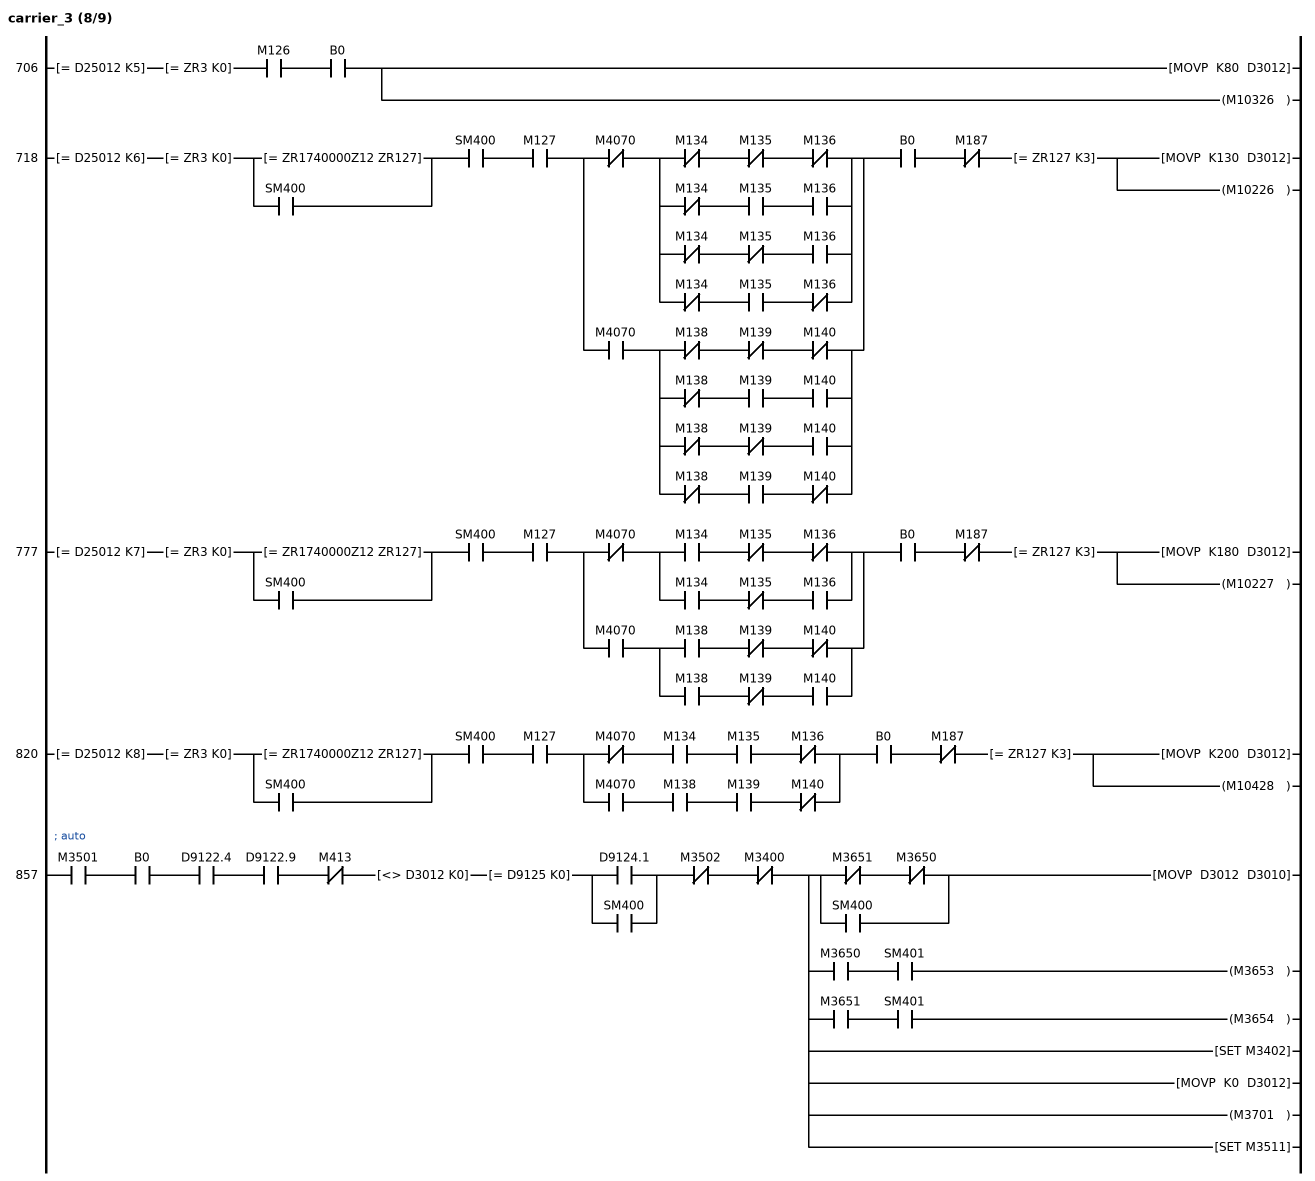
[picture p72: ladder of carrier_3, rungs at steps 706 to 857]
706   LD=     D25012 K5
      AND=    ZR3 K0
      AND     M126
      AND     B0
      MOVP    K80 D3012
      OUT     M10326
718   LD=     D25012 K6
      AND=    ZR3 K0
      LD=     ZR1740000Z12 ZR127
      OR      SM400
      ANB
      AND     SM400
      AND     M127
      LDI     M4070
      LDI     M134
      ANI     M135
      ANI     M136
      LDI     M134
      AND     M135
      AND     M136
      ORB
      LDI     M134
      ANI     M135
      AND     M136
      ORB
      LDI     M134
      AND     M135
      ANI     M136
      ORB
      ANB
      LD      M4070
      LDI     M138
      ANI     M139
      ANI     M140
      LDI     M138
      AND     M139
      AND     M140
      ORB
      LDI     M138
      ANI     M139
      AND     M140
      ORB
      LDI     M138
      AND     M139
      ANI     M140
      ORB
      ANB
      ORB
      ANB
      AND     B0
      ANI     M187
      AND=    ZR127 K3
      MOVP    K130 D3012
      OUT     M10226
777   LD=     D25012 K7
      AND=    ZR3 K0
      LD=     ZR1740000Z12 ZR127
      OR      SM400
      ANB
      AND     SM400
      AND     M127
      LDI     M4070
      LD      M134
      ANI     M135
      ANI     M136
      LD      M134
      ANI     M135
      AND     M136
      ORB
      ANB
      LD      M4070
      LD      M138
      ANI     M139
      ANI     M140
      LD      M138
      ANI     M139
      AND     M140
      ORB
      ANB
      ORB
      ANB
      AND     B0
      ANI     M187
      AND=    ZR127 K3
      MOVP    K180 D3012
      OUT     M10227
820   LD=     D25012 K8
      AND=    ZR3 K0
      LD=     ZR1740000Z12 ZR127
      OR      SM400
      ANB
      AND     SM400
      AND     M127
      LDI     M4070
      AND     M134
      AND     M135
      ANI     M136
      LD      M4070
      AND     M138
      AND     M139
      ANI     M140
      ORB
      ANB
      AND     B0
      ANI     M187
      AND=    ZR127 K3
      MOVP    K200 D3012
      OUT     M10428
; auto
857   LD      M3501
      AND     B0
      AND     D9122.4
      AND     D9122.9
      ANI     M413
      AND<>   D3012 K0
      AND=    D9125 K0
      LD      D9124.1
      OR      SM400
      ANB
      ANI     M3502
      ANI     M3400
      MPS
      LDI     M3651
      ANI     M3650
      OR      SM400
      ANB
      MOVP    D3012 D3010
      MRD
      AND     M3650
      AND     SM401
      OUT     M3653
      MRD
      AND     M3651
      AND     SM401
      OUT     M3654
      MPP
      SET     M3402
      MOVP    K0 D3012
      OUT     M3701
      SET     M3511
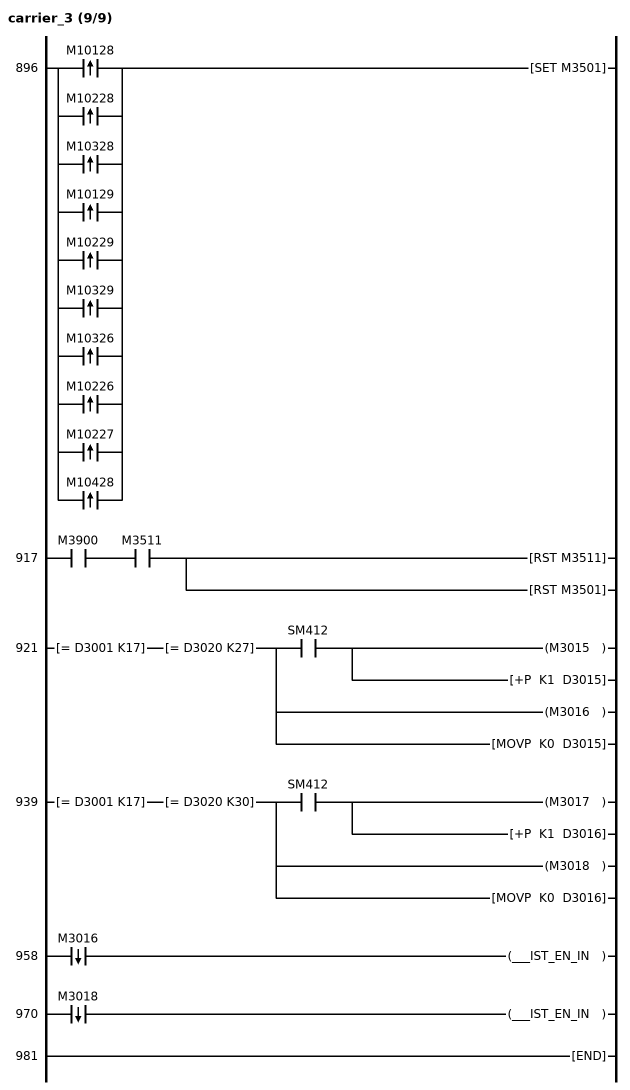
896   LDP     M10128
      ORP     M10228
      ORP     M10328
      ORP     M10129
      ORP     M10229
      ORP     M10329
      ORP     M10326
      ORP     M10226
      ORP     M10227
      ORP     M10428
      SET     M3501
917   LD      M3900
      AND     M3511
      RST     M3511
      RST     M3501
921   LD=     D3001 K17
      AND=    D3020 K27
      MPS
      AND     SM412
      OUT     M3015
      +P      K1 D3015
      MPP
      OUT     M3016
      MOVP    K0 D3015
939   LD=     D3001 K17
      AND=    D3020 K30
      MPS
      AND     SM412
      OUT     M3017
      +P      K1 D3016
      MPP
      OUT     M3018
      MOVP    K0 D3016
; FB BLK START I+ST_76367eaf8b844e8d(__IST_76367eaf8b844e8d)
958   LDF     M3016
      OUT     ___IST_EN_IN
; FB START
; FB_NAME I+ST_76367eaf8b844e8d
; INSTANCE_NAME __IST_76367eaf8b844e8d
; FB IN_B:__IST_EN_IN
; FB OUT___IST_EN_OUT:B
; FB END
; FB BLK END
; FB BLK START I+ST_4f96081e274e4d1c(__IST_4f96081e274e4d1c)
970   LDF     M3018
      OUT     ___IST_EN_IN
; FB START
; FB_NAME I+ST_4f96081e274e4d1c
; INSTANCE_NAME __IST_4f96081e274e4d1c
; FB IN_B:__IST_EN_IN
; FB OUT___IST_EN_OUT:B
; FB END
; FB BLK END
981   END
END_PROGRAM

PROGRAM carrier_4
VAR
  c_comm_4 : c_comm_4;
END_VAR
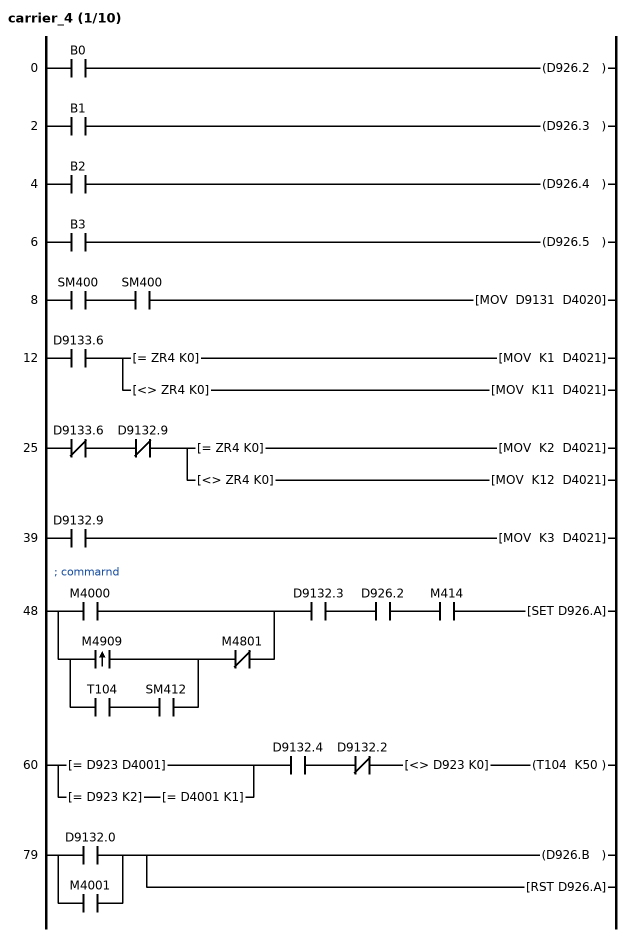
0     LD      B0
      OUT     D926.2
2     LD      B1
      OUT     D926.3
4     LD      B2
      OUT     D926.4
6     LD      B3
      OUT     D926.5
8     LD      SM400
      AND     SM400
      MOV     D9131 D4020
12    LD      D9133.6
      MPS
      AND=    ZR4 K0
      MOV     K1 D4021
      MPP
      AND<>   ZR4 K0
      MOV     K11 D4021
25    LDI     D9133.6
      ANI     D9132.9
      MPS
      AND=    ZR4 K0
      MOV     K2 D4021
      MPP
      AND<>   ZR4 K0
      MOV     K12 D4021
39    LD      D9132.9
      MOV     K3 D4021
; commarnd
48    LD      M4000
      LDP     M4909
      LD      T104
      AND     SM412
      ORB
      ANI     M4801
      ORB
      AND     D9132.3
      AND     D926.2
      AND     M414
      SET     D926.A
60    LD=     D923 D4001
      LD=     D923 K2
      AND=    D4001 K1
      ORB
      AND     D9132.4
      ANI     D9132.2
      AND<>   D923 K0
      OUT     T104 K50
79    LD      D9132.0
      OR      M4001
      OUT     D926.B
      RST     D926.A
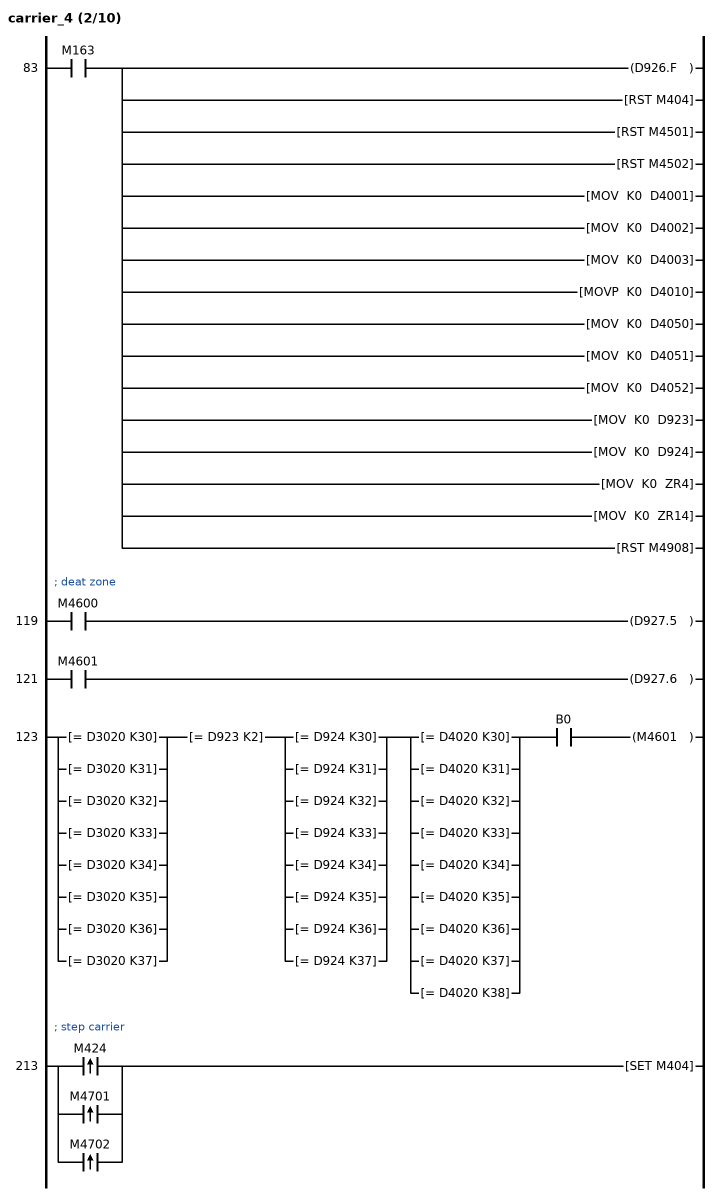
83    LD      M163
      OUT     D926.F
      RST     M404
      RST     M4501
      RST     M4502
      MOV     K0 D4001
      MOV     K0 D4002
      MOV     K0 D4003
      MOVP    K0 D4010
      MOV     K0 D4050
      MOV     K0 D4051
      MOV     K0 D4052
      MOV     K0 D923
      MOV     K0 D924
      MOV     K0 ZR4
      MOV     K0 ZR14
      RST     M4908
; deat zone
119   LD      M4600
      OUT     D927.5
121   LD      M4601
      OUT     D927.6
123   LD=     D3020 K30
      OR=     D3020 K31
      OR=     D3020 K32
      OR=     D3020 K33
      OR=     D3020 K34
      OR=     D3020 K35
      OR=     D3020 K36
      OR=     D3020 K37
      AND=    D923 K2
      LD=     D924 K30
      OR=     D924 K31
      OR=     D924 K32
      OR=     D924 K33
      OR=     D924 K34
      OR=     D924 K35
      OR=     D924 K36
      OR=     D924 K37
      ANB
      LD=     D4020 K30
      OR=     D4020 K31
      OR=     D4020 K32
      OR=     D4020 K33
      OR=     D4020 K34
      OR=     D4020 K35
      OR=     D4020 K36
      OR=     D4020 K37
      OR=     D4020 K38
      ANB
      AND     B0
      OUT     M4601
; step carrier
213   LDP     M424
      ORP     M4701
      ORP     M4702
      SET     M404
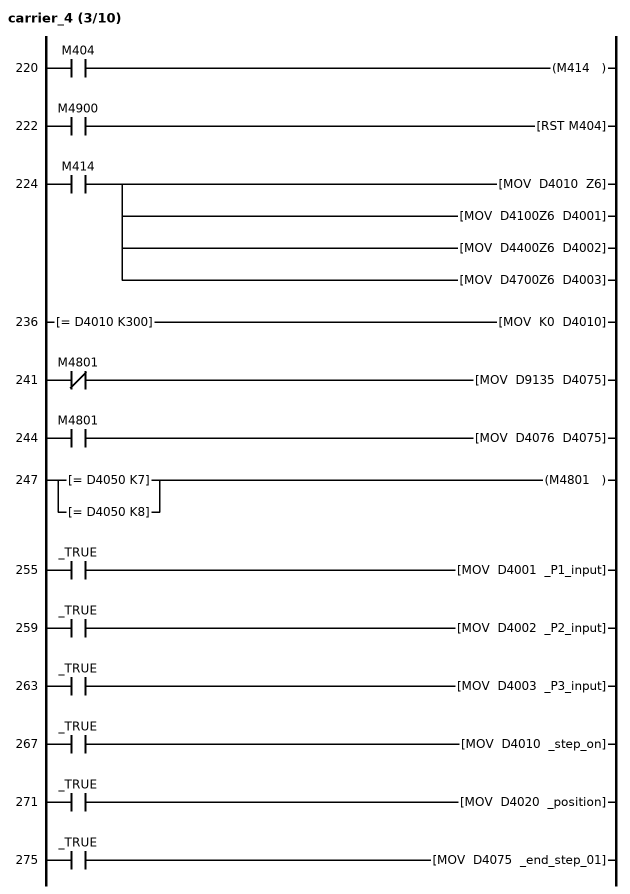
220   LD      M404
      OUT     M414
222   LD      M4900
      RST     M404
224   LD      M414
      MOV     D4010 Z6
      MOV     D4100Z6 D4001
      MOV     D4400Z6 D4002
      MOV     D4700Z6 D4003
236   LD=     D4010 K300
      MOV     K0 D4010
241   LDI     M4801
      MOV     D9135 D4075
244   LD      M4801
      MOV     D4076 D4075
247   LD=     D4050 K7
      OR=     D4050 K8
      OUT     M4801
; FB BLK START c_comm_4(c_comm_4)
255   LD      _TRUE
      MOV     D4001 _P1_input
259   LD      _TRUE
      MOV     D4002 _P2_input
263   LD      _TRUE
      MOV     D4003 _P3_input
267   LD      _TRUE
      MOV     D4010 _step_on
271   LD      _TRUE
      MOV     D4020 _position
275   LD      _TRUE
      MOV     D4075 _end_step_01
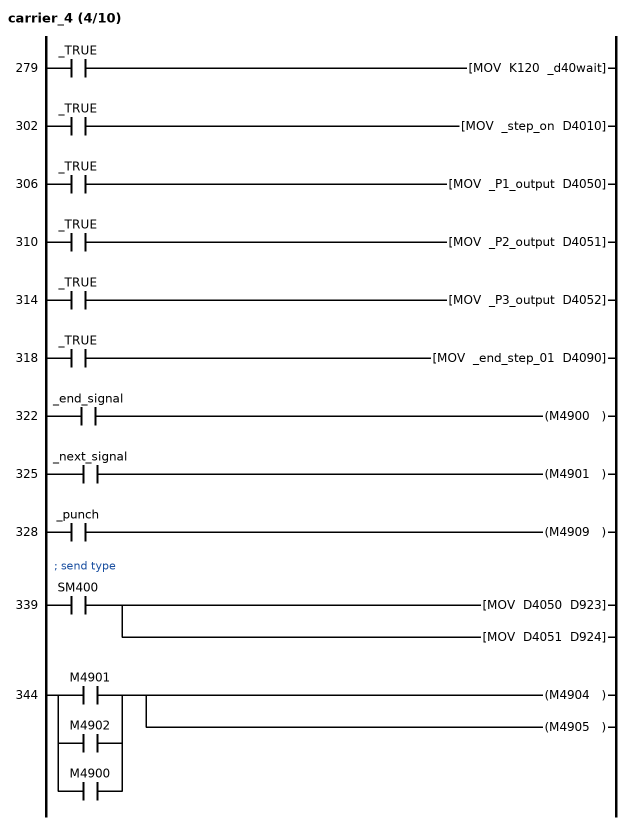
279   LD      _TRUE
      MOV     K120 _d40wait
; FB START
; FB_NAME c_comm_4
; INSTANCE_NAME c_comm_4
; FB IN_W:P1_input
; FB OUT_step_on:W
; FB IN_W:P2_input
; FB OUT_P1_output:W
; FB IN_W:P3_input
; FB OUT_P2_output:W
; FB IN_W:step_on
; FB OUT_P3_output:W
; FB IN_W:position
; FB OUT_end_step_01:W
; FB IN_W:end_step_01
; FB OUT_end_signal:B
; FB IN_W:d40wait
; FB OUT_next_signal:B
; FB OUT_punch:B
; FB END
302   LD      _TRUE
      MOV     _step_on D4010
306   LD      _TRUE
      MOV     _P1_output D4050
310   LD      _TRUE
      MOV     _P2_output D4051
314   LD      _TRUE
      MOV     _P3_output D4052
318   LD      _TRUE
      MOV     _end_step_01 D4090
322   LD      _end_signal
      OUT     M4900
325   LD      _next_signal
      OUT     M4901
328   LD      _punch
      OUT     M4909
; FB BLK END
; send type
339   LD      SM400
      MOV     D4050 D923
      MOV     D4051 D924
344   LD      M4901
      OR      M4902
      OR      M4900
      OUT     M4904
      OUT     M4905
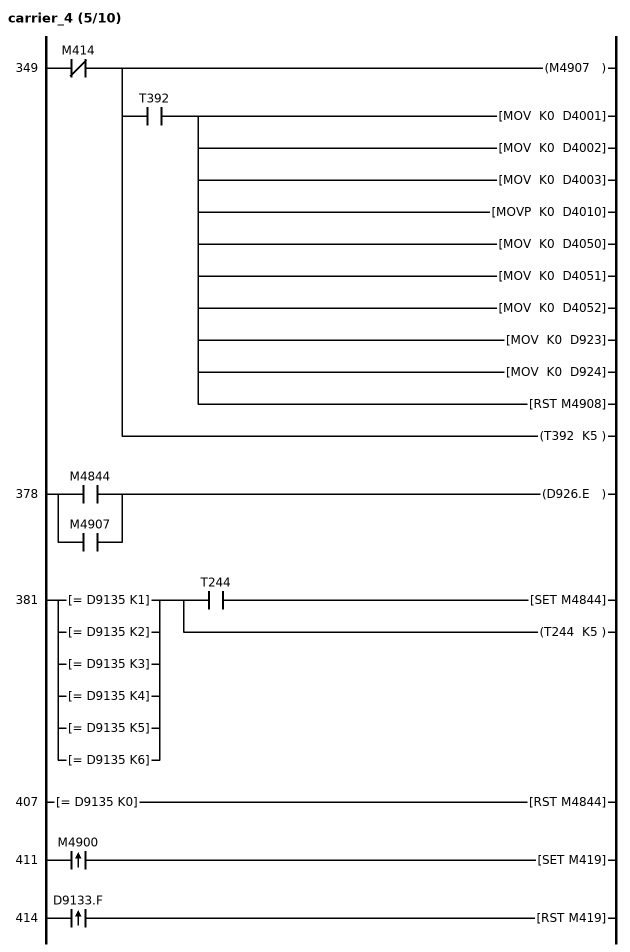
349   LDI     M414
      OUT     M4907
      MPS
      AND     T392
      MOV     K0 D4001
      MOV     K0 D4002
      MOV     K0 D4003
      MOVP    K0 D4010
      MOV     K0 D4050
      MOV     K0 D4051
      MOV     K0 D4052
      MOV     K0 D923
      MOV     K0 D924
      RST     M4908
      MPP
      OUT     T392 K5
378   LD      M4844
      OR      M4907
      OUT     D926.E
381   LD=     D9135 K1
      OR=     D9135 K2
      OR=     D9135 K3
      OR=     D9135 K4
      OR=     D9135 K5
      OR=     D9135 K6
      MPS
      AND     T244
      SET     M4844
      MPP
      OUT     T244 K5
407   LD=     D9135 K0
      RST     M4844
411   LDP     M4900
      SET     M419
414   LDP     D9133.F
      RST     M419
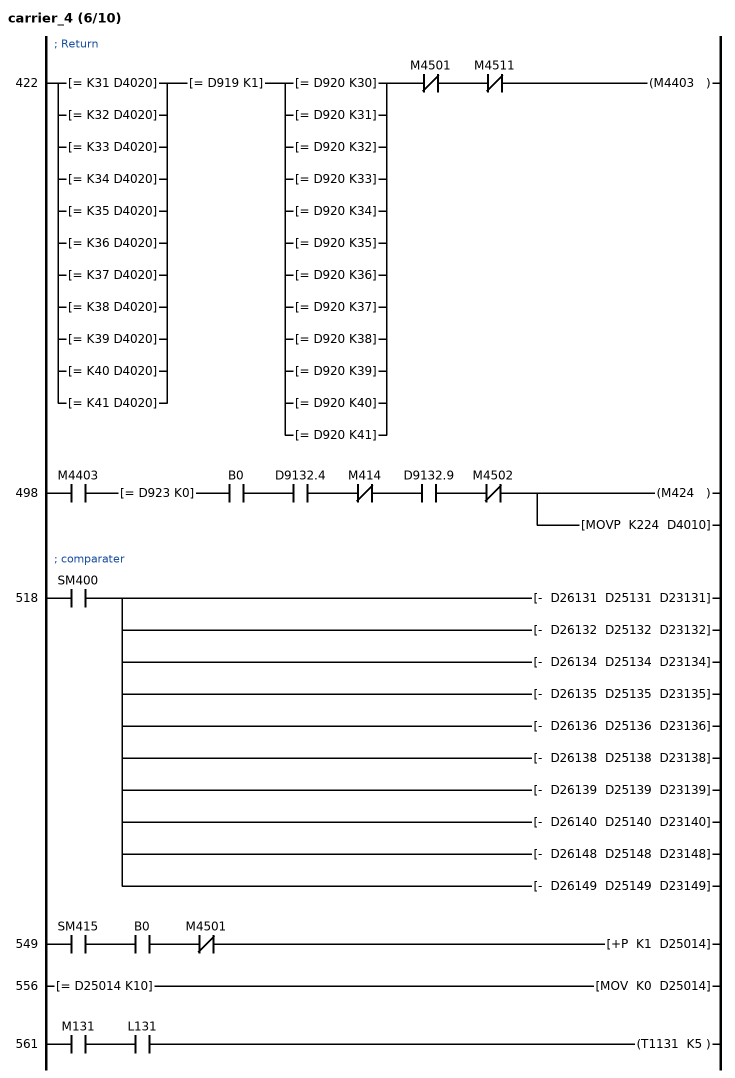
; Return
422   LD=     K31 D4020
      OR=     K32 D4020
      OR=     K33 D4020
      OR=     K34 D4020
      OR=     K35 D4020
      OR=     K36 D4020
      OR=     K37 D4020
      OR=     K38 D4020
      OR=     K39 D4020
      OR=     K40 D4020
      OR=     K41 D4020
      AND=    D919 K1
      LD=     D920 K30
      OR=     D920 K31
      OR=     D920 K32
      OR=     D920 K33
      OR=     D920 K34
      OR=     D920 K35
      OR=     D920 K36
      OR=     D920 K37
      OR=     D920 K38
      OR=     D920 K39
      OR=     D920 K40
      OR=     D920 K41
      ANB
      ANI     M4501
      ANI     M4511
      OUT     M4403
498   LD      M4403
      AND=    D923 K0
      AND     B0
      AND     D9132.4
      ANI     M414
      AND     D9132.9
      ANI     M4502
      OUT     M424
      MOVP    K224 D4010
; comparater
518   LD      SM400
      -       D26131 D25131 D23131
      -       D26132 D25132 D23132
      -       D26134 D25134 D23134
      -       D26135 D25135 D23135
      -       D26136 D25136 D23136
      -       D26138 D25138 D23138
      -       D26139 D25139 D23139
      -       D26140 D25140 D23140
      -       D26148 D25148 D23148
      -       D26149 D25149 D23149
549   LD      SM415
      AND     B0
      ANI     M4501
      +P      K1 D25014
556   LD=     D25014 K10
      MOV     K0 D25014
561   LD      M131
      AND     L131
      OUT     T1131 K5
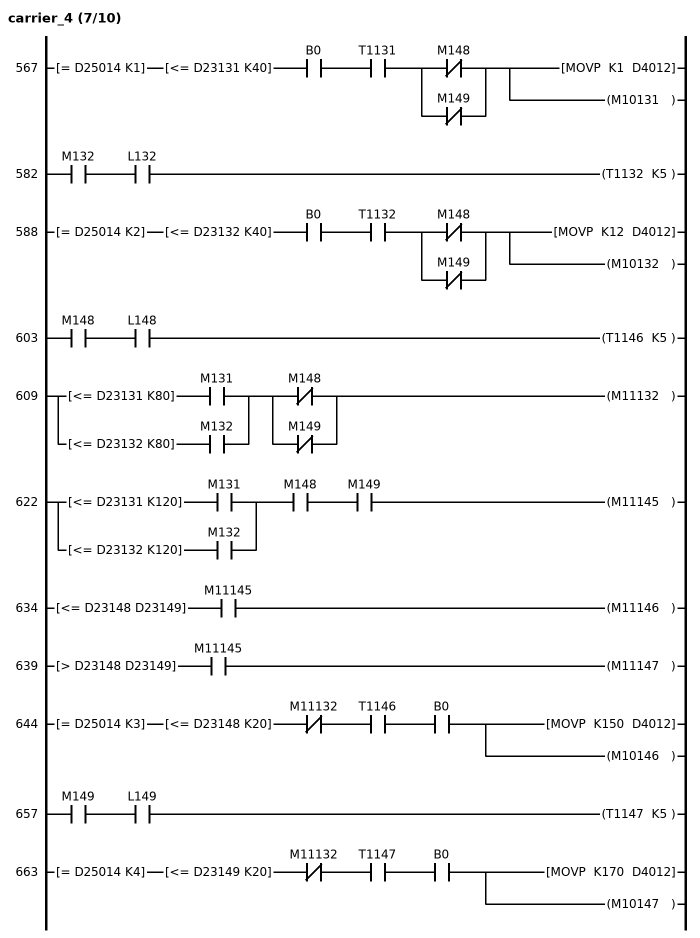
567   LD=     D25014 K1
      AND<=   D23131 K40
      AND     B0
      AND     T1131
      LDI     M148
      ORI     M149
      ANB
      MOVP    K1 D4012
      OUT     M10131
582   LD      M132
      AND     L132
      OUT     T1132 K5
588   LD=     D25014 K2
      AND<=   D23132 K40
      AND     B0
      AND     T1132
      LDI     M148
      ORI     M149
      ANB
      MOVP    K12 D4012
      OUT     M10132
603   LD      M148
      AND     L148
      OUT     T1146 K5
609   LD<=    D23131 K80
      AND     M131
      LD<=    D23132 K80
      AND     M132
      ORB
      LDI     M148
      ORI     M149
      ANB
      OUT     M11132
622   LD<=    D23131 K120
      AND     M131
      LD<=    D23132 K120
      AND     M132
      ORB
      AND     M148
      AND     M149
      OUT     M11145
634   LD<=    D23148 D23149
      AND     M11145
      OUT     M11146
639   LD>     D23148 D23149
      AND     M11145
      OUT     M11147
644   LD=     D25014 K3
      AND<=   D23148 K20
      ANI     M11132
      AND     T1146
      AND     B0
      MOVP    K150 D4012
      OUT     M10146
657   LD      M149
      AND     L149
      OUT     T1147 K5
663   LD=     D25014 K4
      AND<=   D23149 K20
      ANI     M11132
      AND     T1147
      AND     B0
      MOVP    K170 D4012
      OUT     M10147
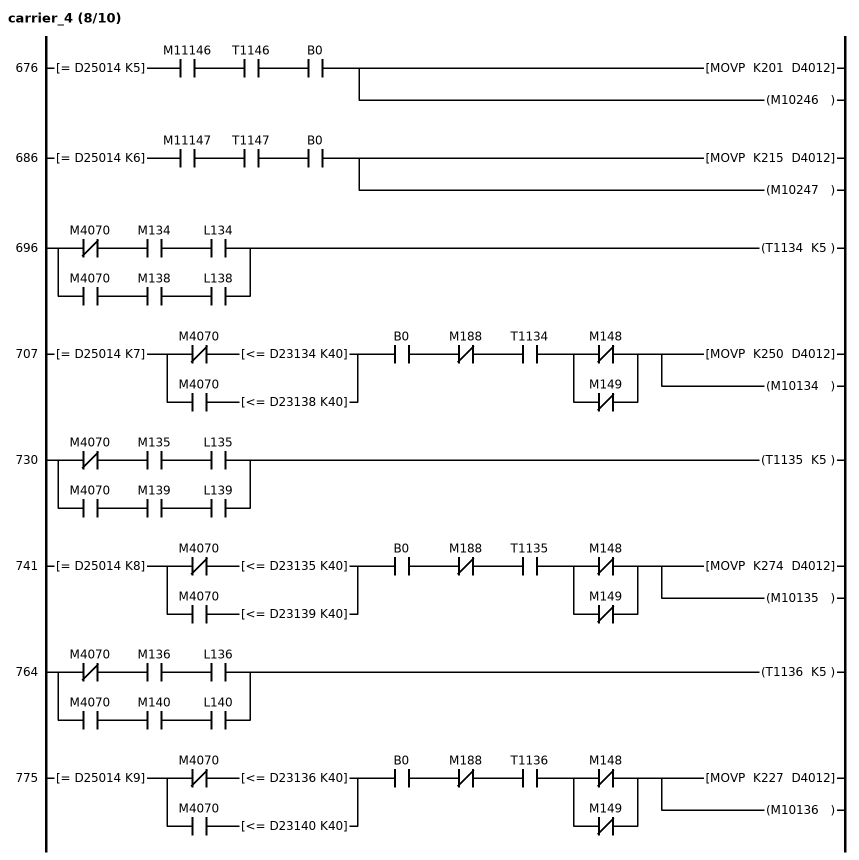
676   LD=     D25014 K5
      AND     M11146
      AND     T1146
      AND     B0
      MOVP    K201 D4012
      OUT     M10246
686   LD=     D25014 K6
      AND     M11147
      AND     T1147
      AND     B0
      MOVP    K215 D4012
      OUT     M10247
696   LDI     M4070
      AND     M134
      AND     L134
      LD      M4070
      AND     M138
      AND     L138
      ORB
      OUT     T1134 K5
707   LD=     D25014 K7
      LDI     M4070
      AND<=   D23134 K40
      LD      M4070
      AND<=   D23138 K40
      ORB
      ANB
      AND     B0
      ANI     M188
      AND     T1134
      LDI     M148
      ORI     M149
      ANB
      MOVP    K250 D4012
      OUT     M10134
730   LDI     M4070
      AND     M135
      AND     L135
      LD      M4070
      AND     M139
      AND     L139
      ORB
      OUT     T1135 K5
741   LD=     D25014 K8
      LDI     M4070
      AND<=   D23135 K40
      LD      M4070
      AND<=   D23139 K40
      ORB
      ANB
      AND     B0
      ANI     M188
      AND     T1135
      LDI     M148
      ORI     M149
      ANB
      MOVP    K274 D4012
      OUT     M10135
764   LDI     M4070
      AND     M136
      AND     L136
      LD      M4070
      AND     M140
      AND     L140
      ORB
      OUT     T1136 K5
775   LD=     D25014 K9
      LDI     M4070
      AND<=   D23136 K40
      LD      M4070
      AND<=   D23140 K40
      ORB
      ANB
      AND     B0
      ANI     M188
      AND     T1136
      LDI     M148
      ORI     M149
      ANB
      MOVP    K227 D4012
      OUT     M10136
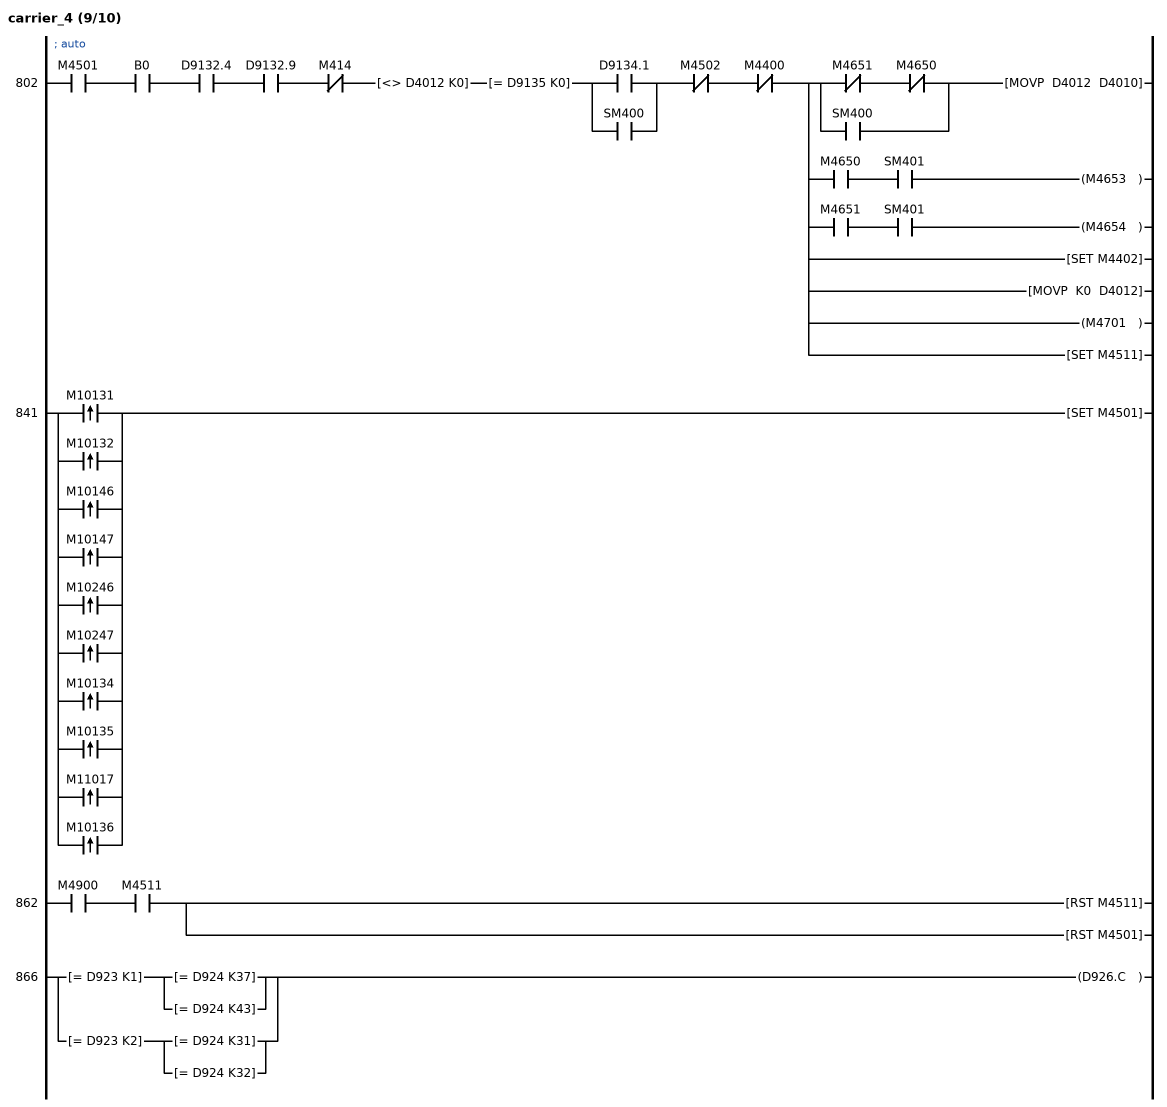
; auto
802   LD      M4501
      AND     B0
      AND     D9132.4
      AND     D9132.9
      ANI     M414
      AND<>   D4012 K0
      AND=    D9135 K0
      LD      D9134.1
      OR      SM400
      ANB
      ANI     M4502
      ANI     M4400
      MPS
      LDI     M4651
      ANI     M4650
      OR      SM400
      ANB
      MOVP    D4012 D4010
      MRD
      AND     M4650
      AND     SM401
      OUT     M4653
      MRD
      AND     M4651
      AND     SM401
      OUT     M4654
      MPP
      SET     M4402
      MOVP    K0 D4012
      OUT     M4701
      SET     M4511
841   LDP     M10131
      ORP     M10132
      ORP     M10146
      ORP     M10147
      ORP     M10246
      ORP     M10247
      ORP     M10134
      ORP     M10135
      ORP     M11017
      ORP     M10136
      SET     M4501
862   LD      M4900
      AND     M4511
      RST     M4511
      RST     M4501
866   LD=     D923 K1
      LD=     D924 K37
      OR=     D924 K43
      ANB
      LD=     D923 K2
      LD=     D924 K31
      OR=     D924 K32
      ANB
      ORB
      OUT     D926.C
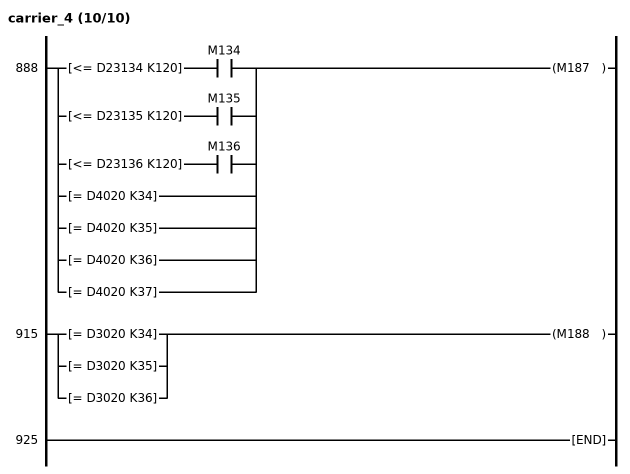
888   LD<=    D23134 K120
      AND     M134
      LD<=    D23135 K120
      AND     M135
      ORB
      LD<=    D23136 K120
      AND     M136
      ORB
      OR=     D4020 K34
      OR=     D4020 K35
      OR=     D4020 K36
      OR=     D4020 K37
      OUT     M187
915   LD=     D3020 K34
      OR=     D3020 K35
      OR=     D3020 K36
      OUT     M188
925   END
END_PROGRAM

PROGRAM carrier_reset
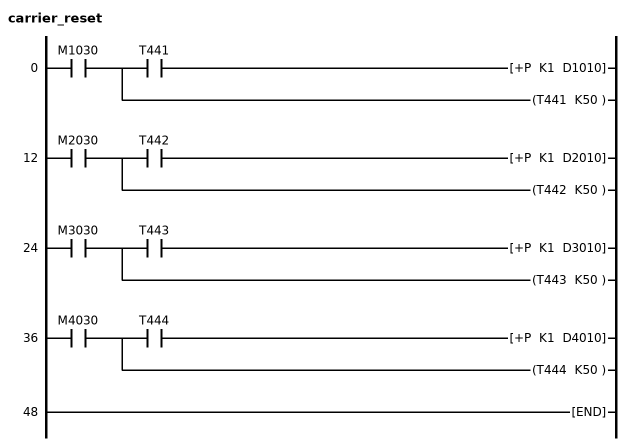
0     LD      M1030
      MPS
      AND     T441
      +P      K1 D1010
      MPP
      OUT     T441 K50
12    LD      M2030
      MPS
      AND     T442
      +P      K1 D2010
      MPP
      OUT     T442 K50
24    LD      M3030
      MPS
      AND     T443
      +P      K1 D3010
      MPP
      OUT     T443 K50
36    LD      M4030
      MPS
      AND     T444
      +P      K1 D4010
      MPP
      OUT     T444 K50
48    END
END_PROGRAM

PROGRAM couter
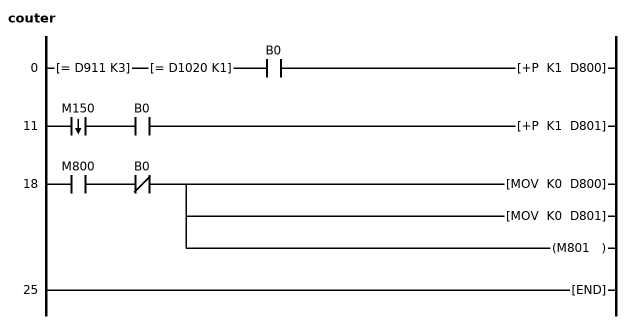
0     LD=     D911 K3
      AND=    D1020 K1
      AND     B0
      +P      K1 D800
11    LDF     M150
      AND     B0
      +P      K1 D801
18    LD      M800
      ANI     B0
      MOV     K0 D800
      MOV     K0 D801
      OUT     M801
25    END
END_PROGRAM

PROGRAM data_carry
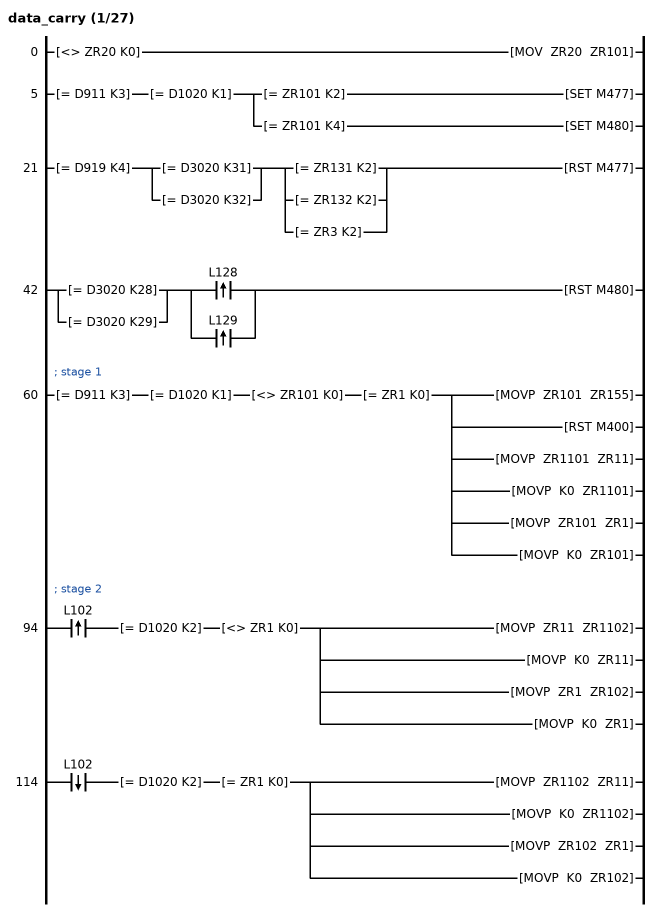
0     LD<>    ZR20 K0
      MOV     ZR20 ZR101
5     LD=     D911 K3
      AND=    D1020 K1
      MPS
      AND=    ZR101 K2
      SET     M477
      MPP
      AND=    ZR101 K4
      SET     M480
21    LD=     D919 K4
      LD=     D3020 K31
      OR=     D3020 K32
      ANB
      LD=     ZR131 K2
      OR=     ZR132 K2
      OR=     ZR3 K2
      ANB
      RST     M477
42    LD=     D3020 K28
      OR=     D3020 K29
      LDP     L128
      ORP     L129
      ANB
      RST     M480
; stage 1
60    LD=     D911 K3
      AND=    D1020 K1
      AND<>   ZR101 K0
      AND=    ZR1 K0
      MOVP    ZR101 ZR155
      RST     M400
      MOVP    ZR1101 ZR11
      MOVP    K0 ZR1101
      MOVP    ZR101 ZR1
      MOVP    K0 ZR101
; stage 2
94    LDP     L102
      AND=    D1020 K2
      AND<>   ZR1 K0
      MOVP    ZR11 ZR1102
      MOVP    K0 ZR11
      MOVP    ZR1 ZR102
      MOVP    K0 ZR1
114   LDF     L102
      AND=    D1020 K2
      AND=    ZR1 K0
      MOVP    ZR1102 ZR11
      MOVP    K0 ZR1102
      MOVP    ZR102 ZR1
      MOVP    K0 ZR102
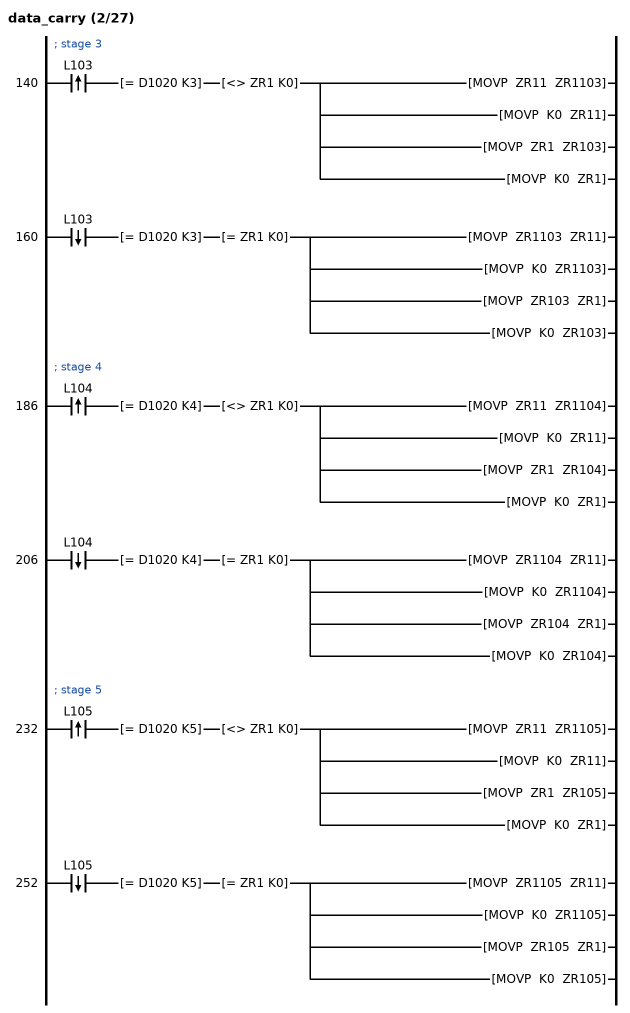
; stage 3
140   LDP     L103
      AND=    D1020 K3
      AND<>   ZR1 K0
      MOVP    ZR11 ZR1103
      MOVP    K0 ZR11
      MOVP    ZR1 ZR103
      MOVP    K0 ZR1
160   LDF     L103
      AND=    D1020 K3
      AND=    ZR1 K0
      MOVP    ZR1103 ZR11
      MOVP    K0 ZR1103
      MOVP    ZR103 ZR1
      MOVP    K0 ZR103
; stage 4
186   LDP     L104
      AND=    D1020 K4
      AND<>   ZR1 K0
      MOVP    ZR11 ZR1104
      MOVP    K0 ZR11
      MOVP    ZR1 ZR104
      MOVP    K0 ZR1
206   LDF     L104
      AND=    D1020 K4
      AND=    ZR1 K0
      MOVP    ZR1104 ZR11
      MOVP    K0 ZR1104
      MOVP    ZR104 ZR1
      MOVP    K0 ZR104
; stage 5
232   LDP     L105
      AND=    D1020 K5
      AND<>   ZR1 K0
      MOVP    ZR11 ZR1105
      MOVP    K0 ZR11
      MOVP    ZR1 ZR105
      MOVP    K0 ZR1
252   LDF     L105
      AND=    D1020 K5
      AND=    ZR1 K0
      MOVP    ZR1105 ZR11
      MOVP    K0 ZR1105
      MOVP    ZR105 ZR1
      MOVP    K0 ZR105
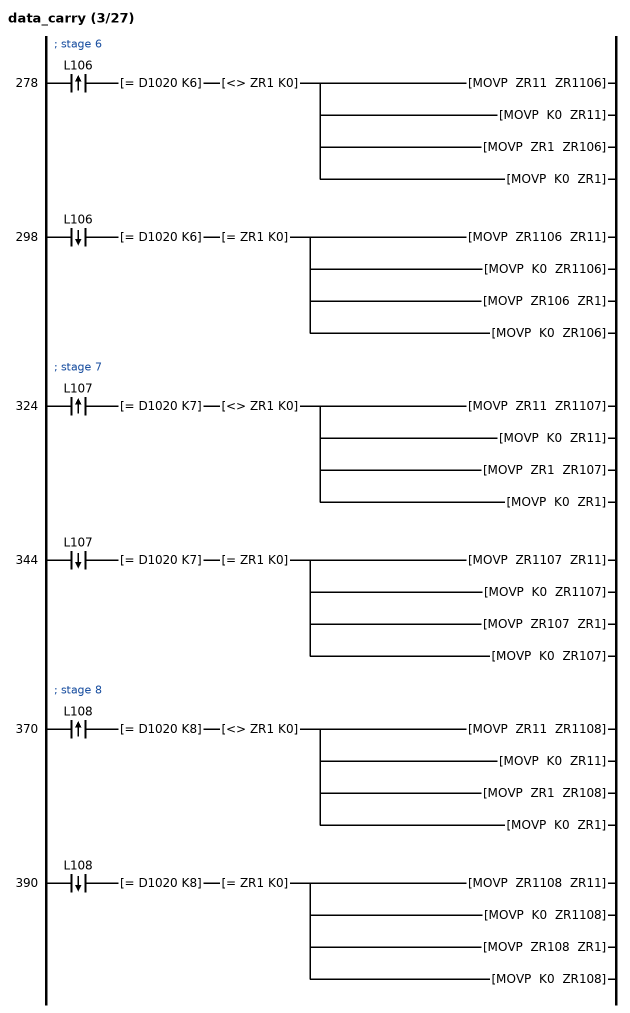
; stage 6
278   LDP     L106
      AND=    D1020 K6
      AND<>   ZR1 K0
      MOVP    ZR11 ZR1106
      MOVP    K0 ZR11
      MOVP    ZR1 ZR106
      MOVP    K0 ZR1
298   LDF     L106
      AND=    D1020 K6
      AND=    ZR1 K0
      MOVP    ZR1106 ZR11
      MOVP    K0 ZR1106
      MOVP    ZR106 ZR1
      MOVP    K0 ZR106
; stage 7
324   LDP     L107
      AND=    D1020 K7
      AND<>   ZR1 K0
      MOVP    ZR11 ZR1107
      MOVP    K0 ZR11
      MOVP    ZR1 ZR107
      MOVP    K0 ZR1
344   LDF     L107
      AND=    D1020 K7
      AND=    ZR1 K0
      MOVP    ZR1107 ZR11
      MOVP    K0 ZR1107
      MOVP    ZR107 ZR1
      MOVP    K0 ZR107
; stage 8
370   LDP     L108
      AND=    D1020 K8
      AND<>   ZR1 K0
      MOVP    ZR11 ZR1108
      MOVP    K0 ZR11
      MOVP    ZR1 ZR108
      MOVP    K0 ZR1
390   LDF     L108
      AND=    D1020 K8
      AND=    ZR1 K0
      MOVP    ZR1108 ZR11
      MOVP    K0 ZR1108
      MOVP    ZR108 ZR1
      MOVP    K0 ZR108
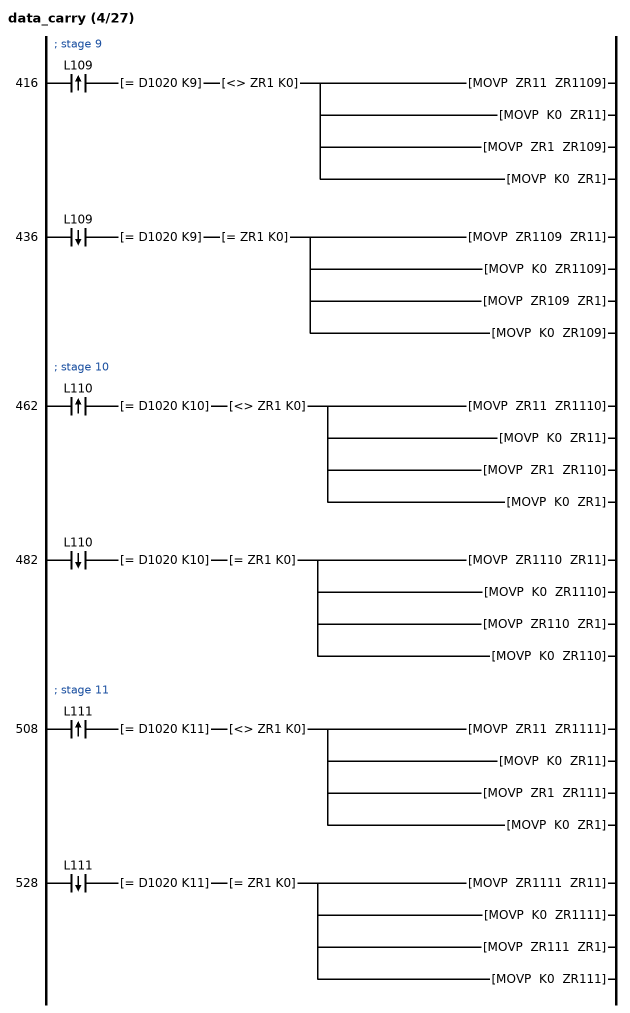
; stage 9
416   LDP     L109
      AND=    D1020 K9
      AND<>   ZR1 K0
      MOVP    ZR11 ZR1109
      MOVP    K0 ZR11
      MOVP    ZR1 ZR109
      MOVP    K0 ZR1
436   LDF     L109
      AND=    D1020 K9
      AND=    ZR1 K0
      MOVP    ZR1109 ZR11
      MOVP    K0 ZR1109
      MOVP    ZR109 ZR1
      MOVP    K0 ZR109
; stage 10
462   LDP     L110
      AND=    D1020 K10
      AND<>   ZR1 K0
      MOVP    ZR11 ZR1110
      MOVP    K0 ZR11
      MOVP    ZR1 ZR110
      MOVP    K0 ZR1
482   LDF     L110
      AND=    D1020 K10
      AND=    ZR1 K0
      MOVP    ZR1110 ZR11
      MOVP    K0 ZR1110
      MOVP    ZR110 ZR1
      MOVP    K0 ZR110
; stage 11
508   LDP     L111
      AND=    D1020 K11
      AND<>   ZR1 K0
      MOVP    ZR11 ZR1111
      MOVP    K0 ZR11
      MOVP    ZR1 ZR111
      MOVP    K0 ZR1
528   LDF     L111
      AND=    D1020 K11
      AND=    ZR1 K0
      MOVP    ZR1111 ZR11
      MOVP    K0 ZR1111
      MOVP    ZR111 ZR1
      MOVP    K0 ZR111
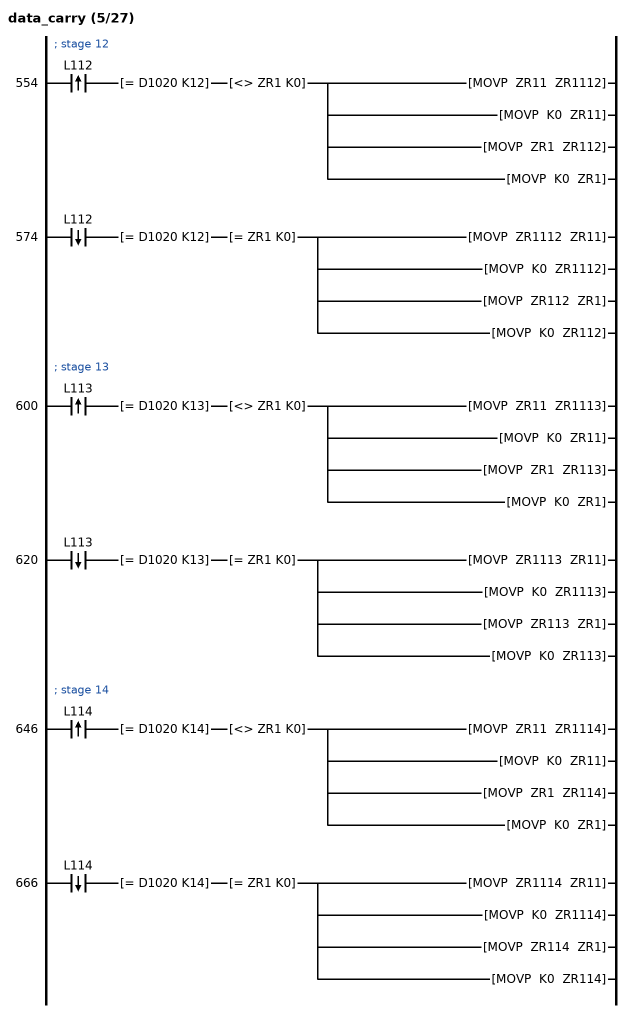
; stage 12
554   LDP     L112
      AND=    D1020 K12
      AND<>   ZR1 K0
      MOVP    ZR11 ZR1112
      MOVP    K0 ZR11
      MOVP    ZR1 ZR112
      MOVP    K0 ZR1
574   LDF     L112
      AND=    D1020 K12
      AND=    ZR1 K0
      MOVP    ZR1112 ZR11
      MOVP    K0 ZR1112
      MOVP    ZR112 ZR1
      MOVP    K0 ZR112
; stage 13
600   LDP     L113
      AND=    D1020 K13
      AND<>   ZR1 K0
      MOVP    ZR11 ZR1113
      MOVP    K0 ZR11
      MOVP    ZR1 ZR113
      MOVP    K0 ZR1
620   LDF     L113
      AND=    D1020 K13
      AND=    ZR1 K0
      MOVP    ZR1113 ZR11
      MOVP    K0 ZR1113
      MOVP    ZR113 ZR1
      MOVP    K0 ZR113
; stage 14
646   LDP     L114
      AND=    D1020 K14
      AND<>   ZR1 K0
      MOVP    ZR11 ZR1114
      MOVP    K0 ZR11
      MOVP    ZR1 ZR114
      MOVP    K0 ZR1
666   LDF     L114
      AND=    D1020 K14
      AND=    ZR1 K0
      MOVP    ZR1114 ZR11
      MOVP    K0 ZR1114
      MOVP    ZR114 ZR1
      MOVP    K0 ZR114
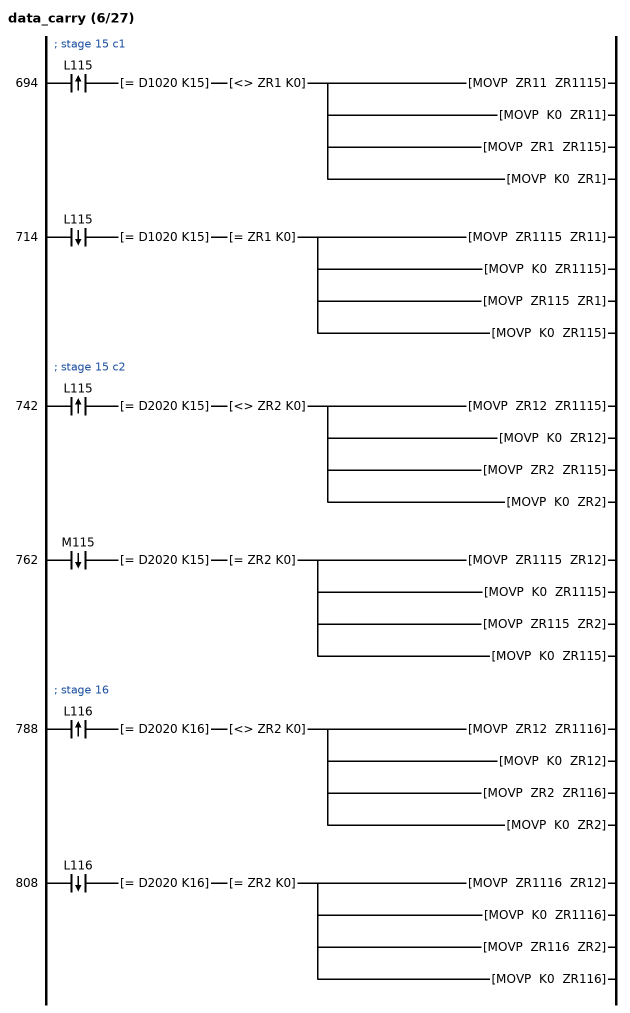
; stage 15 c1
694   LDP     L115
      AND=    D1020 K15
      AND<>   ZR1 K0
      MOVP    ZR11 ZR1115
      MOVP    K0 ZR11
      MOVP    ZR1 ZR115
      MOVP    K0 ZR1
714   LDF     L115
      AND=    D1020 K15
      AND=    ZR1 K0
      MOVP    ZR1115 ZR11
      MOVP    K0 ZR1115
      MOVP    ZR115 ZR1
      MOVP    K0 ZR115
; stage 15 c2
742   LDP     L115
      AND=    D2020 K15
      AND<>   ZR2 K0
      MOVP    ZR12 ZR1115
      MOVP    K0 ZR12
      MOVP    ZR2 ZR115
      MOVP    K0 ZR2
762   LDF     M115
      AND=    D2020 K15
      AND=    ZR2 K0
      MOVP    ZR1115 ZR12
      MOVP    K0 ZR1115
      MOVP    ZR115 ZR2
      MOVP    K0 ZR115
; stage 16
788   LDP     L116
      AND=    D2020 K16
      AND<>   ZR2 K0
      MOVP    ZR12 ZR1116
      MOVP    K0 ZR12
      MOVP    ZR2 ZR116
      MOVP    K0 ZR2
808   LDF     L116
      AND=    D2020 K16
      AND=    ZR2 K0
      MOVP    ZR1116 ZR12
      MOVP    K0 ZR1116
      MOVP    ZR116 ZR2
      MOVP    K0 ZR116
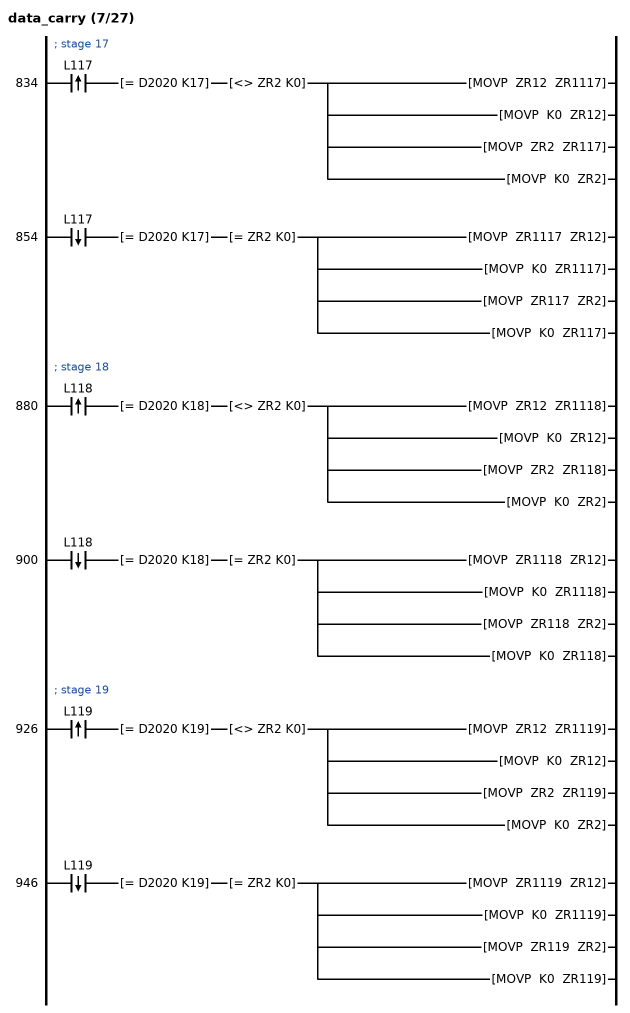
; stage 17
834   LDP     L117
      AND=    D2020 K17
      AND<>   ZR2 K0
      MOVP    ZR12 ZR1117
      MOVP    K0 ZR12
      MOVP    ZR2 ZR117
      MOVP    K0 ZR2
854   LDF     L117
      AND=    D2020 K17
      AND=    ZR2 K0
      MOVP    ZR1117 ZR12
      MOVP    K0 ZR1117
      MOVP    ZR117 ZR2
      MOVP    K0 ZR117
; stage 18
880   LDP     L118
      AND=    D2020 K18
      AND<>   ZR2 K0
      MOVP    ZR12 ZR1118
      MOVP    K0 ZR12
      MOVP    ZR2 ZR118
      MOVP    K0 ZR2
900   LDF     L118
      AND=    D2020 K18
      AND=    ZR2 K0
      MOVP    ZR1118 ZR12
      MOVP    K0 ZR1118
      MOVP    ZR118 ZR2
      MOVP    K0 ZR118
; stage 19
926   LDP     L119
      AND=    D2020 K19
      AND<>   ZR2 K0
      MOVP    ZR12 ZR1119
      MOVP    K0 ZR12
      MOVP    ZR2 ZR119
      MOVP    K0 ZR2
946   LDF     L119
      AND=    D2020 K19
      AND=    ZR2 K0
      MOVP    ZR1119 ZR12
      MOVP    K0 ZR1119
      MOVP    ZR119 ZR2
      MOVP    K0 ZR119
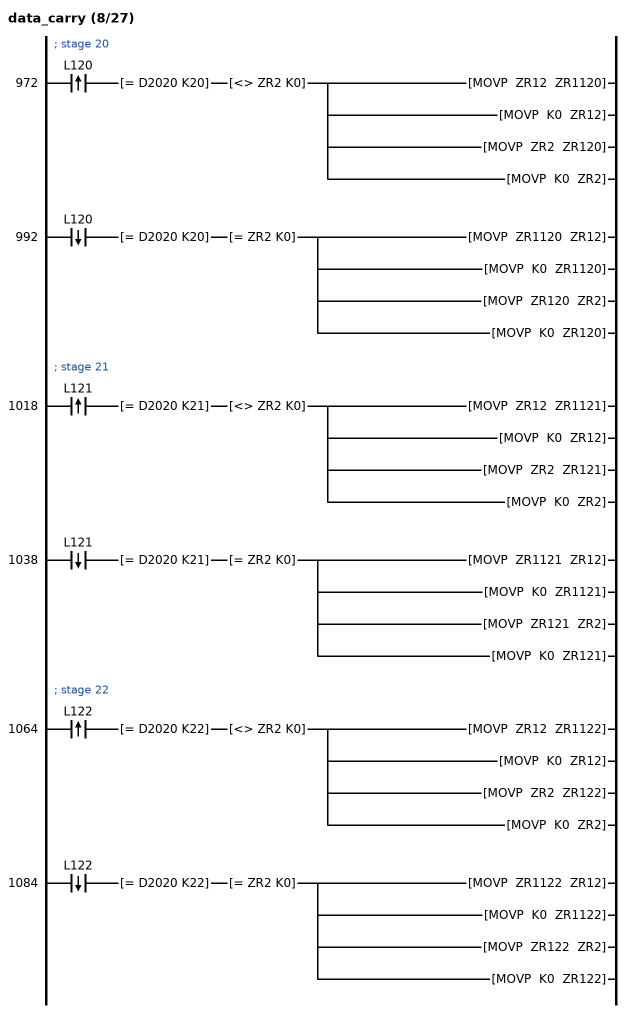
; stage 20
972   LDP     L120
      AND=    D2020 K20
      AND<>   ZR2 K0
      MOVP    ZR12 ZR1120
      MOVP    K0 ZR12
      MOVP    ZR2 ZR120
      MOVP    K0 ZR2
992   LDF     L120
      AND=    D2020 K20
      AND=    ZR2 K0
      MOVP    ZR1120 ZR12
      MOVP    K0 ZR1120
      MOVP    ZR120 ZR2
      MOVP    K0 ZR120
; stage 21
1018  LDP     L121
      AND=    D2020 K21
      AND<>   ZR2 K0
      MOVP    ZR12 ZR1121
      MOVP    K0 ZR12
      MOVP    ZR2 ZR121
      MOVP    K0 ZR2
1038  LDF     L121
      AND=    D2020 K21
      AND=    ZR2 K0
      MOVP    ZR1121 ZR12
      MOVP    K0 ZR1121
      MOVP    ZR121 ZR2
      MOVP    K0 ZR121
; stage 22
1064  LDP     L122
      AND=    D2020 K22
      AND<>   ZR2 K0
      MOVP    ZR12 ZR1122
      MOVP    K0 ZR12
      MOVP    ZR2 ZR122
      MOVP    K0 ZR2
1084  LDF     L122
      AND=    D2020 K22
      AND=    ZR2 K0
      MOVP    ZR1122 ZR12
      MOVP    K0 ZR1122
      MOVP    ZR122 ZR2
      MOVP    K0 ZR122
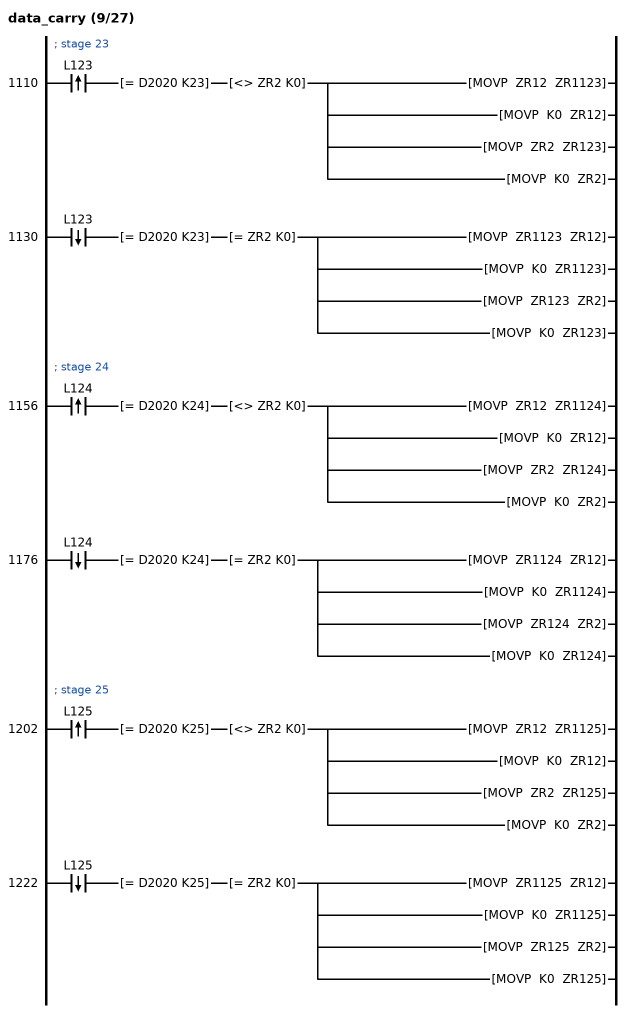
; stage 23
1110  LDP     L123
      AND=    D2020 K23
      AND<>   ZR2 K0
      MOVP    ZR12 ZR1123
      MOVP    K0 ZR12
      MOVP    ZR2 ZR123
      MOVP    K0 ZR2
1130  LDF     L123
      AND=    D2020 K23
      AND=    ZR2 K0
      MOVP    ZR1123 ZR12
      MOVP    K0 ZR1123
      MOVP    ZR123 ZR2
      MOVP    K0 ZR123
; stage 24
1156  LDP     L124
      AND=    D2020 K24
      AND<>   ZR2 K0
      MOVP    ZR12 ZR1124
      MOVP    K0 ZR12
      MOVP    ZR2 ZR124
      MOVP    K0 ZR2
1176  LDF     L124
      AND=    D2020 K24
      AND=    ZR2 K0
      MOVP    ZR1124 ZR12
      MOVP    K0 ZR1124
      MOVP    ZR124 ZR2
      MOVP    K0 ZR124
; stage 25
1202  LDP     L125
      AND=    D2020 K25
      AND<>   ZR2 K0
      MOVP    ZR12 ZR1125
      MOVP    K0 ZR12
      MOVP    ZR2 ZR125
      MOVP    K0 ZR2
1222  LDF     L125
      AND=    D2020 K25
      AND=    ZR2 K0
      MOVP    ZR1125 ZR12
      MOVP    K0 ZR1125
      MOVP    ZR125 ZR2
      MOVP    K0 ZR125
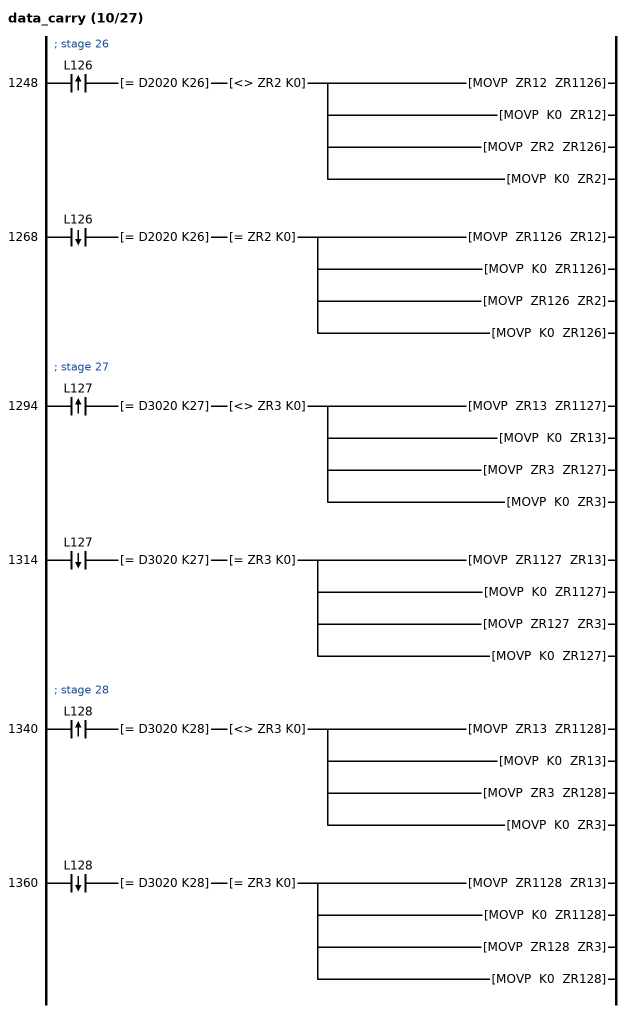
; stage 26
1248  LDP     L126
      AND=    D2020 K26
      AND<>   ZR2 K0
      MOVP    ZR12 ZR1126
      MOVP    K0 ZR12
      MOVP    ZR2 ZR126
      MOVP    K0 ZR2
1268  LDF     L126
      AND=    D2020 K26
      AND=    ZR2 K0
      MOVP    ZR1126 ZR12
      MOVP    K0 ZR1126
      MOVP    ZR126 ZR2
      MOVP    K0 ZR126
; stage 27
1294  LDP     L127
      AND=    D3020 K27
      AND<>   ZR3 K0
      MOVP    ZR13 ZR1127
      MOVP    K0 ZR13
      MOVP    ZR3 ZR127
      MOVP    K0 ZR3
1314  LDF     L127
      AND=    D3020 K27
      AND=    ZR3 K0
      MOVP    ZR1127 ZR13
      MOVP    K0 ZR1127
      MOVP    ZR127 ZR3
      MOVP    K0 ZR127
; stage 28
1340  LDP     L128
      AND=    D3020 K28
      AND<>   ZR3 K0
      MOVP    ZR13 ZR1128
      MOVP    K0 ZR13
      MOVP    ZR3 ZR128
      MOVP    K0 ZR3
1360  LDF     L128
      AND=    D3020 K28
      AND=    ZR3 K0
      MOVP    ZR1128 ZR13
      MOVP    K0 ZR1128
      MOVP    ZR128 ZR3
      MOVP    K0 ZR128
